TYPE TcoDiConfig :
STRUCT
    IsFalseTimeOut : TIME := T#10S;
    IsTrueTimeOut : TIME := T#10S;
END_STRUCT
END_TYPE

(* stored: Version 1.1.0.1
   DUT TcoDiConfig: Id {81cad678-50b3-0c03-09c5-050fe48ae5b3} *)
